TYPE ST_BaseLocationDesctription :
STRUCT
	wsDescription		: WSTRING;
	sCade				: STRING;
END_STRUCT
END_TYPE

(* stored: Version 1.1.0.1
   DUT ST_BaseLocationDesctription: Id {1af1b441-63c2-0606-1554-fb8c58ce1fee} *)
